KUKA KRL data list: $config.dat

&ACCESS RV$1
DEFDAT $CONFIG

ENDDAT
